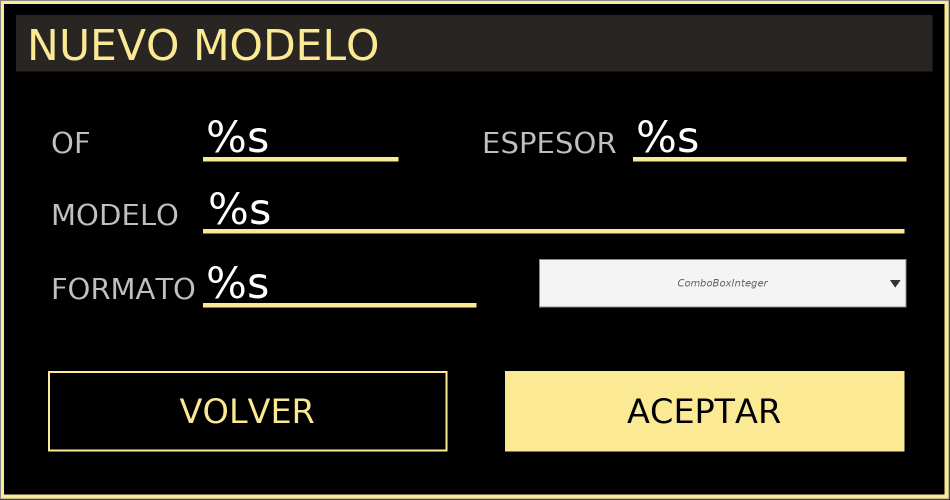
VISUALIZATION Modelo_Tabla_Md2  // 950x500
    Rectangle (0,0 948x498)
    Rectangle (424,1281 690x58), "%s Contador piezas Multidiscos 2", text variable: FuncParoNodoMultidiscos.Funci_Multidiscos2.Cont_Piezas_Ftc
    Button (1159,1261 269x91), "Reset contador"
        tap FuncParoNodoMultidiscos.Funci_Multidiscos2.Pul_Reset_Cnt_Piez
    ComboBoxInteger (539,259 367x48), variable: FuncParoNodoMultidiscos.FunGeneMultidiscos2.IndexListFormatoTabla, text list: 'FormatoTabla'
    Rectangle (16,15 916x56)
    Label (24,17 498x56), "NUEVO MODELO"
    Rectangle (205,185 701x48), "%s", text variable: FuncParoNodoMultidiscos.FunGeneMultidiscos2.s_ModeloEleccionTabla
        OnMouseDown: write the text variable via Edit
    Label (48,197 148x36), "MODELO"
    Rectangle (203,229 701x4)
    Rectangle (203,259 273x48), "%s", text variable: FuncParoNodoMultidiscos.FunGeneMultidiscos2.s_FormatoEleccionTabla, input disabled if: FuncParoNodoMultidiscos.FunGeneMultidiscos2.IndexListFormatoTabla<>0
        OnMouseDown: write the text variable via Edit
    Label (48,271 148x36), "FORMATO"
    Rectangle (203,303 273x4)
    Rectangle (633,113 273x48), "%s", text variable: FuncParoNodoMultidiscos.FunGeneMultidiscos2.s_EspesorEleccionTabla
        OnMouseDown: write the text variable via Edit
    Label (479,125 148x36), "ESPESOR"
    Rectangle (633,157 273x4)
    Rectangle (505,371 399x80), "ACEPTAR"
        tap FuncParoNodoMultidiscos.FunGeneMultidiscos2.P_EscribirModelo
        OnMouseClick: CloseDialog Dialog=Modelo_Tabla_Md2, Result=OK, NumpadKeypadSet=True
    Rectangle (48,371 399x80), "VOLVER"
        OnMouseClick: CloseDialog Dialog=Modelo_Tabla_Md2, Result=Cancel, NumpadKeypadSet=True
    Group (48,113 350x48)
        Rectangle (155,0 195x48), "%s", text variable: FuncParoNodoCorteH4Remote1.sEspesorActualTabla
            OnMouseDown: write the text variable via Edit
        Label (0,12 148x36), "OF"
        Rectangle (155,44 195x4)
END_VISUALIZATION

(* stored: Version 1.1.0.1, ProductVersion 3.1.4024.12
   Visu Modelo_Tabla_Md2: Id {39aa03c3-fde9-4505-8c37-4d34977e9f24} *)
